// TIA Portal V17 export
// export: Created 2025-11-28T12:28:54.5679296Z, ExportSetting WithDefaults, WithReadOnly, DisplayName Totally Integrated Automation Portal, DisplayVersion V17 Update 7, DisplayName TIA Portal Openness, DisplayVersion V17 Update 7, DisplayName TIA Portal Version Control Interface, DisplayVersion V17, DisplayName SINAMICS Startdrive Advanced, DisplayVersion V17 SP2, DisplayName SINAMICS DCC, DisplayVersion V17 Update 1, DisplayName SINAMICS Startdrive G110M, G120, G120C, G120D, G120P, G115D, DisplayVersion V17 SP2, DisplayName SINAMICS Startdrive G130, G150, S120, S150, SINAMICS MV, S210, DisplayVersion V17 SP2, DisplayName STEP 7 Professional, DisplayVersion V17 Update 7, DisplayName STEP 7 Safety, DisplayVersion V17 Update 6, DisplayName WinCC Advanced, DisplayVersion V17 Update 7, DisplayName SIMATIC Visualization Architect, DisplayVersion V17 Update 7
FUNCTION "[nome_FC]" : Void   // FC[numero_FC], LAD
TITLE = Rob_[nome_robo]
{ S7_Optimized_Access := 'TRUE' }
VERSION : 1.1
// stored: AutoNumber false, CodeModifiedDate 2024-11-12T14:50:14.9301897Z, CompileDate 2024-11-12T14:50:14.9301897Z, CreationDate 2024-09-18T08:44:27.9878747Z, HandleErrorsWithinBlock false, InterfaceModifiedDate 2017-06-20T14:56:01.2096118Z, IsConsistent true, IsIECCheckEnabled false, IsKnowHowProtected false, IsWriteProtected false, LibraryConformanceStatus Error: The block contains calls of single instances. Warning: The object contains access to global data blocks. Warning: The block contains direct access to inputs, outputs, bit memories, indirect access to the registry or indirect access to external memory areas that are unknown at the time of compilation., ModifiedDate 2024-11-12T14:50:14.9301897Z, ParameterModified 2017-06-20T14:56:01.2021118Z, PLCSimAdvancedSupport true, SetENOAutomatically false, StructureModified 2017-06-20T14:56:01.2096118Z, UDAEnableTagReadback false
   VAR_TEMP
      Temp : Struct
         _Bool : Bool;
         _Byte : Byte;
         _Word : Word;
         _DWord : DWord;
         _Int : Int;
         _DInt : DInt;
         _Real : Real;
         _S5Time : S5Time;
         _Time : Time;
      END_STRUCT;
   END_VAR
BEGIN
END_FUNCTION
